Fanuc KAREL source: kc00008.KL

-- PROVISIONAL review KL for V940-1; original PC SHA256 bf237988952e678f9666b52306efe3a71f7d43c7ad32c9cebda09932f4fb1498
-- Incomplete behavior may be omitted. Consult companion uncertainty JSON. Do not deploy.
PROGRAM KC00008
%NOLOCKGROUP
BEGIN
  -- V9_ZERO_TABLE_METADATA_HINT layout=0002_ascii; no indexed target words; source/name/runtime held
  -- UNRESOLVED_PC offsets 5-33; opcodes 27,22,1C,22,22,31
  -- UNRESOLVED_PC offsets 38-42; opcodes 7F
END KC00008
